// TIA Portal V20 export
VAR_GLOBAL   // PLC tag table "SPREADER"
   iMainLoadPin1In AT %IW600 : Int;   // Main load pin 1
   iMainLoadPin2In AT %IW602 : Int;   // Main load pin 2
   iMainLoadPin3In AT %IW604 : Int;   // Main load pin 3
   iMainLoadPin4In AT %IW606 : Int;   // Main load pin 4
   iRedundantLoadPin1In AT %IW608 : Int;   // Redundant load pin 1
   iRedundantLoadPin2In AT %IW610 : Int;   // Redundant load pin 2
   iRedundantLoadPin3In AT %IW612 : Int;   // Redundant load pin 3
   iRedundantLoadPin4In AT %IW614 : Int;   // Redundant load pin 4
END_VAR
